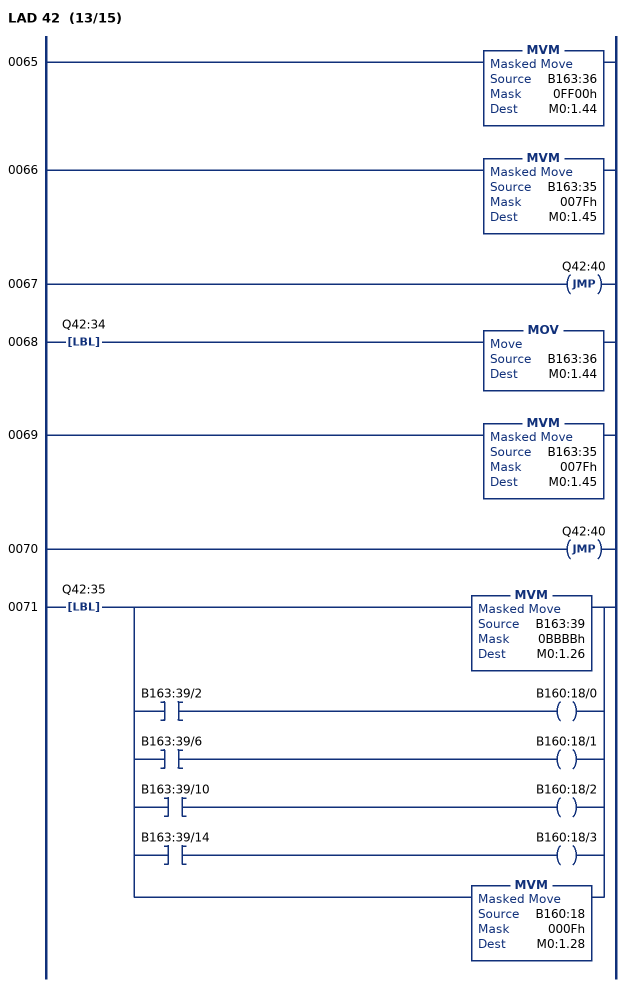
% Rung: 65 %
SOR MVM B163:36 0FF00h M0:1.44 EOR
% Rung: 66 %
SOR MVM B163:35 007Fh M0:1.45 EOR
% Rung: 67 %
SOR JMP Q42:40 EOR
% Rung: 68 %
SOR LBL Q42:34 MOV B163:36 M0:1.44 EOR
% Rung: 69 %
SOR MVM B163:35 007Fh M0:1.45 EOR
% Rung: 70 %
SOR JMP Q42:40 EOR
% Rung: 71 %
SOR LBL Q42:35 BST MVM B163:39 0BBBBh M0:1.26 NXB XIC B163:39/2 OTE B160:18/0 NXB XIC B163:39/6 OTE B160:18/1 NXB XIC B163:39/10 OTE B160:18/2 NXB XIC B163:39/14 OTE B160:18/3 NXB MVM B160:18 000Fh M0:1.28 BND EOR

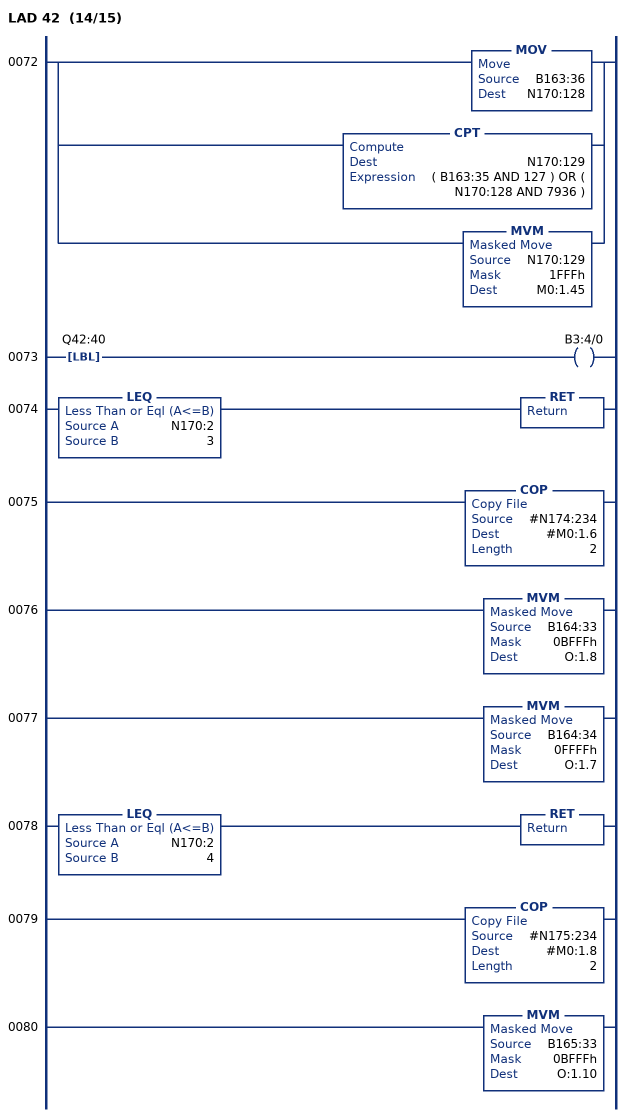
% Rung: 72 %
SOR BST MOV B163:36 N170:128 NXB CPT N170:129 " ( B163:35 AND 127 ) OR ( N170:128 AND 7936 ) " NXB MVM N170:129 1FFFh M0:1.45 BND EOR
% Rung: 73 %
SOR LBL Q42:40 OTE B3:4/0 EOR
% Rung: 74 %
SOR LEQ N170:2 3 RET EOR
% Rung: 75 %
SOR COP #N174:234 #M0:1.6 2 EOR
% Rung: 76 %
SOR MVM B164:33 0BFFFh O:1.8 EOR
% Rung: 77 %
SOR MVM B164:34 0FFFFh O:1.7 EOR
% Rung: 78 %
SOR LEQ N170:2 4 RET EOR
% Rung: 79 %
SOR COP #N175:234 #M0:1.8 2 EOR
% Rung: 80 %
SOR MVM B165:33 0BFFFh O:1.10 EOR

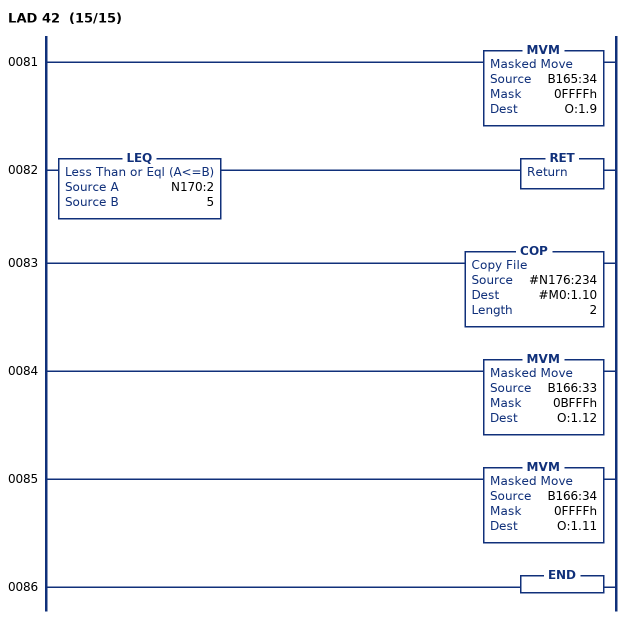
% Rung: 81 %
SOR MVM B165:34 0FFFFh O:1.9 EOR
% Rung: 82 %
SOR LEQ N170:2 5 RET EOR
% Rung: 83 %
SOR COP #N176:234 #M0:1.10 2 EOR
% Rung: 84 %
SOR MVM B166:33 0BFFFh O:1.12 EOR
% Rung: 85 %
SOR MVM B166:34 0FFFFh O:1.11 EOR
% Rung: 86 %
SOR END EOR

LADDER 43
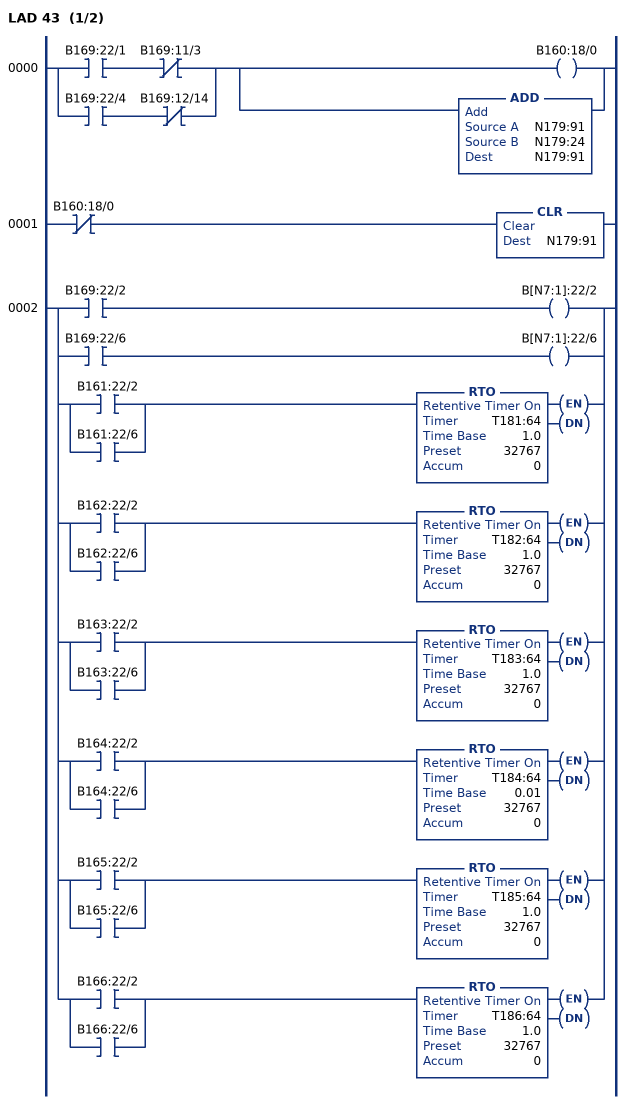
% Rung: 0 %
SOR BST XIC B169:22/1 XIO B169:11/3 NXB XIC B169:22/4 XIO B169:12/14 BND BST OTE B160:18/0 NXB ADD N179:91 N179:24 N179:91 BND EOR
% Rung: 1 %
SOR XIO B160:18/0 CLR N179:91 EOR
% Rung: 2 %
SOR BST BST XIC B169:22/2 OTE B[N7:1]:22/2 NXB XIC B169:22/6 OTE B[N7:1]:22/6 BND NXB BST XIC B161:22/2 NXB XIC B161:22/6 BND RTO T181:64 1.0 32767 0 NXB BST XIC B162:22/2 NXB XIC B162:22/6 BND RTO T182:64 1.0 32767 0 NXB BST XIC B163:22/2 NXB XIC B163:22/6 BND RTO T183:64 1.0 32767 0 NXB BST XIC B164:22/2 NXB XIC B164:22/6 BND RTO T184:64 0.01 32767 0 NXB BST XIC B165:22/2 NXB XIC B165:22/6 BND RTO T185:64 1.0 32767 0 NXB BST XIC B166:22/2 NXB XIC B166:22/6 BND RTO T186:64 1.0 32767 0 BND EOR

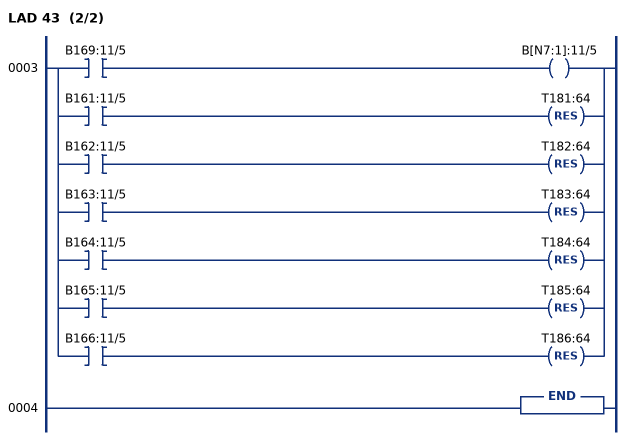
% Rung: 3 %
SOR BST XIC B169:11/5 OTE B[N7:1]:11/5 NXB XIC B161:11/5 RES T181:64 NXB XIC B162:11/5 RES T182:64 NXB XIC B163:11/5 RES T183:64 NXB XIC B164:11/5 RES T184:64 NXB XIC B165:11/5 RES T185:64 NXB XIC B166:11/5 RES T186:64 BND EOR
% Rung: 4 %
SOR END EOR

LADDER 44
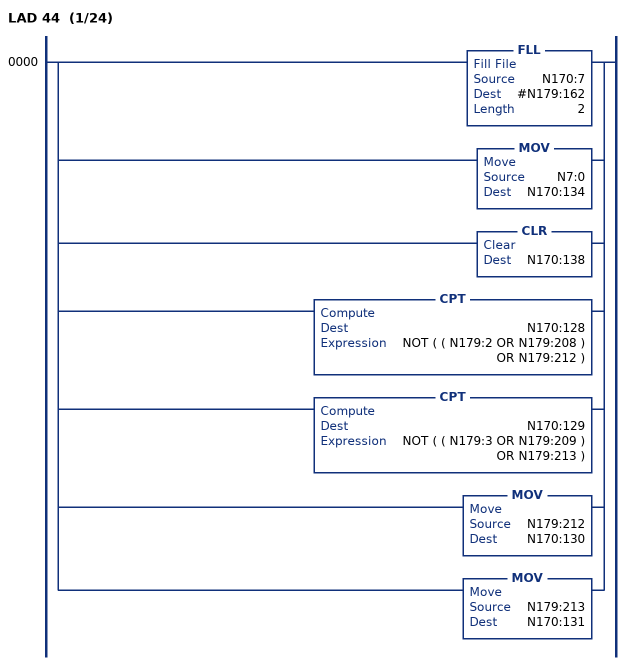
% Rung: 0 %
SOR BST FLL N170:7 #N179:162 2 NXB MOV N7:0 N170:134 NXB CLR N170:138 NXB CPT N170:128 " NOT ( ( N179:2 OR N179:208 ) OR N179:212 ) " NXB CPT N170:129 " NOT ( ( N179:3 OR N179:209 ) OR N179:213 ) " NXB MOV N179:212 N170:130 NXB MOV N179:213 N170:131 BND EOR

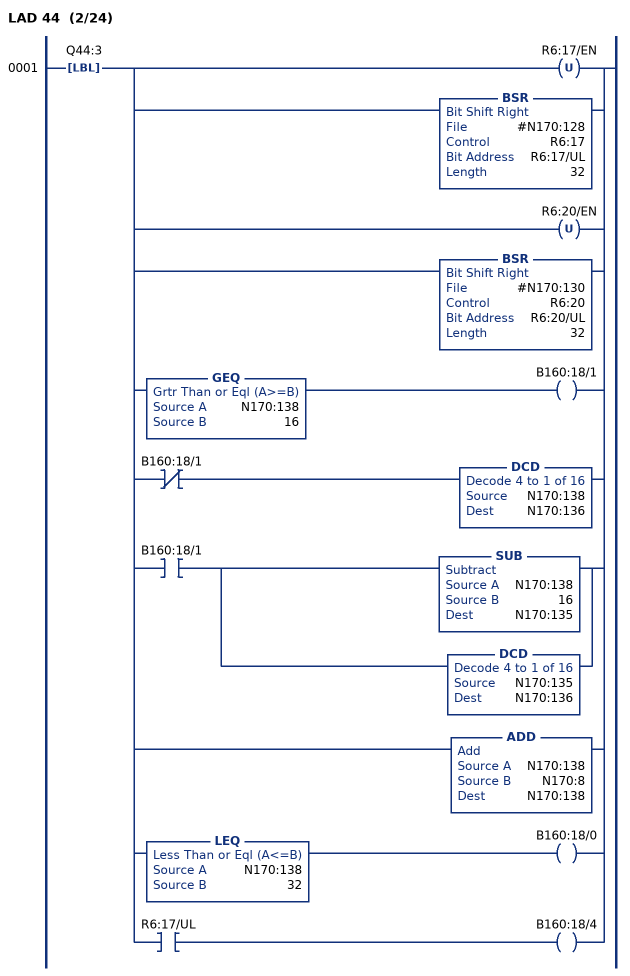
% Rung: 1 %
SOR LBL Q44:3 BST BST OTU R6:17/EN NXB BSR #N170:128 R6:17 R6:17/UL 32 BND NXB BST OTU R6:20/EN NXB BSR #N170:130 R6:20 R6:20/UL 32 BND NXB GEQ N170:138 16 OTE B160:18/1 NXB XIO B160:18/1 DCD N170:138 N170:136 NXB XIC B160:18/1 BST SUB N170:138 16 N170:135 NXB DCD N170:135 N170:136 BND NXB ADD N170:138 N170:8 N170:138 NXB LEQ N170:138 32 OTE B160:18/0 NXB XIC R6:17/UL OTE B160:18/4 BND EOR

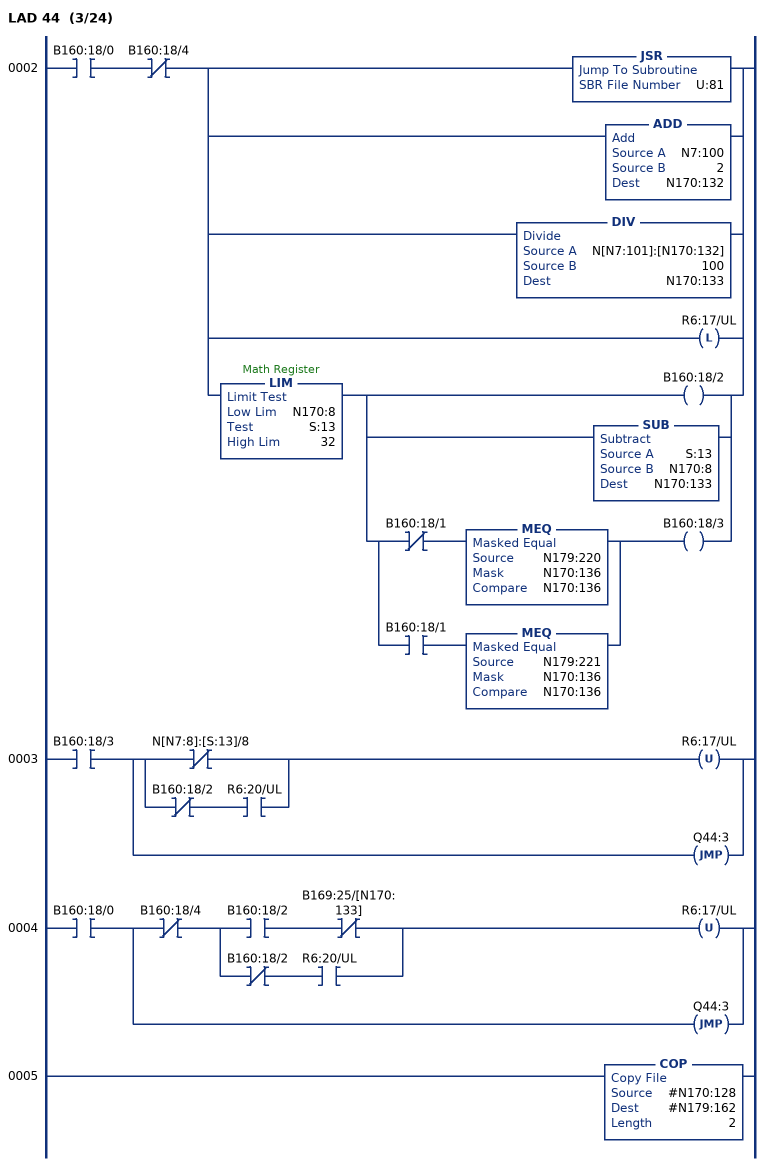
% Rung: 2 %
SOR XIC B160:18/0 XIO B160:18/4 BST JSR U:81 NXB ADD N7:100 2 N170:132 NXB DIV N[N7:101]:[N170:132] 100 N170:133 NXB OTL R6:17/UL NXB LIM N170:8 S:13 32 BST OTE B160:18/2 NXB SUB S:13 N170:8 N170:133 NXB BST XIO B160:18/1 MEQ N179:220 N170:136 N170:136 NXB XIC B160:18/1 MEQ N179:221 N170:136 N170:136 BND OTE B160:18/3 BND BND EOR
%   S:13  "Math Register" %
% Rung: 3 %
SOR XIC B160:18/3 BST BST XIO N[N7:8]:[S:13]/8 NXB XIO B160:18/2 XIC R6:20/UL BND OTU R6:17/UL NXB JMP Q44:3 BND EOR
%   S:13  "Math Register" %
% Rung: 4 %
SOR XIC B160:18/0 BST XIO B160:18/4 BST XIC B160:18/2 XIO B169:25/[N170:133] NXB XIO B160:18/2 XIC R6:20/UL BND OTU R6:17/UL NXB JMP Q44:3 BND EOR
% Rung: 5 %
SOR COP #N170:128 #N179:162 2 EOR

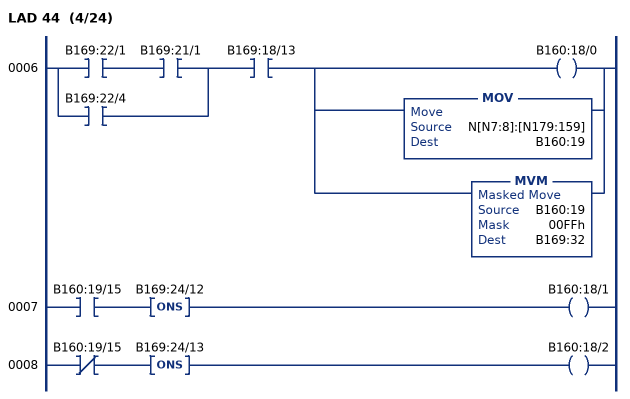
% Rung: 6 %
SOR BST XIC B169:22/1 XIC B169:21/1 NXB XIC B169:22/4 BND XIC B169:18/13 BST OTE B160:18/0 NXB MOV N[N7:8]:[N179:159] B160:19 NXB MVM B160:19 00FFh B169:32 BND EOR
% Rung: 7 %
SOR XIC B160:19/15 OSR B169:24/12 OTE B160:18/1 EOR
% Rung: 8 %
SOR XIO B160:19/15 OSR B169:24/13 OTE B160:18/2 EOR

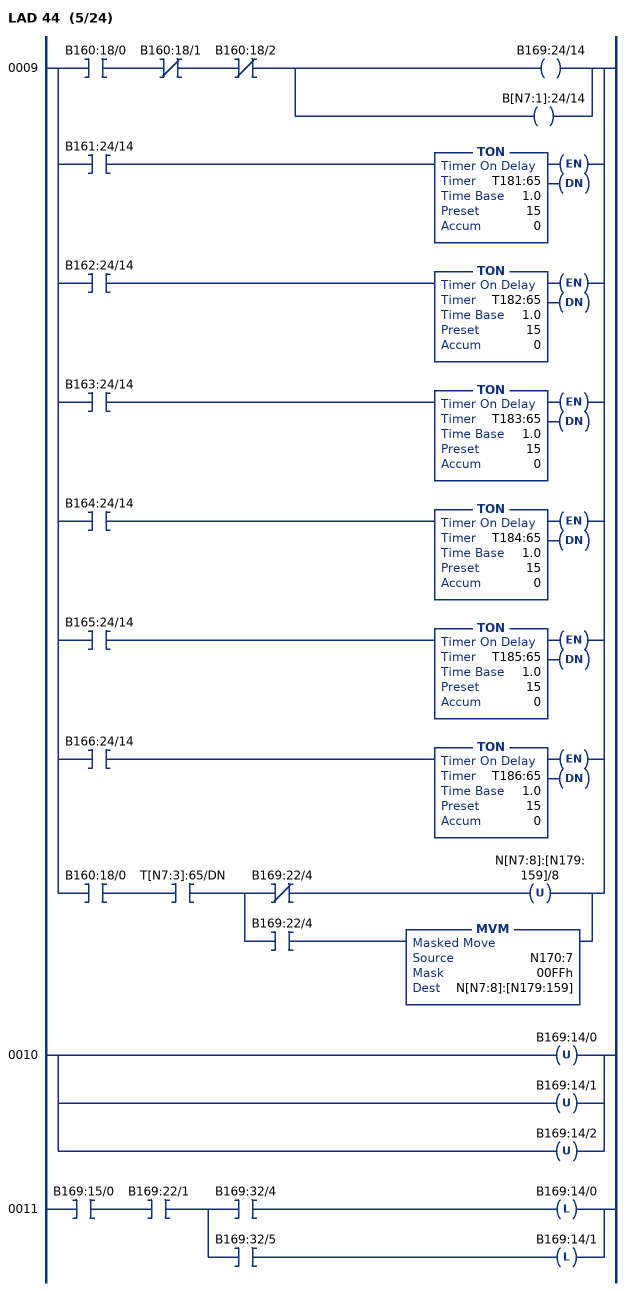
% Rung: 9 %
SOR BST BST XIC B160:18/0 XIO B160:18/1 XIO B160:18/2 BST OTE B169:24/14 NXB OTE B[N7:1]:24/14 BND NXB XIC B161:24/14 TON T181:65 1.0 15 0 NXB XIC B162:24/14 TON T182:65 1.0 15 0 NXB XIC B163:24/14 TON T183:65 1.0 15 0 NXB XIC B164:24/14 TON T184:65 1.0 15 0 NXB XIC B165:24/14 TON T185:65 1.0 15 0 NXB XIC B166:24/14 TON T186:65 1.0 15 0 BND NXB XIC B160:18/0 XIC T[N7:3]:65/DN BST XIO B169:22/4 OTU N[N7:8]:[N179:159]/8 NXB XIC B169:22/4 MVM N170:7 00FFh N[N7:8]:[N179:159] BND BND EOR
% Rung: 10 %
SOR BST OTU B169:14/0 NXB OTU B169:14/1 NXB OTU B169:14/2 BND EOR
% Rung: 11 %
SOR XIC B169:15/0 XIC B169:22/1 BST XIC B169:32/4 OTL B169:14/0 NXB XIC B169:32/5 OTL B169:14/1 BND EOR

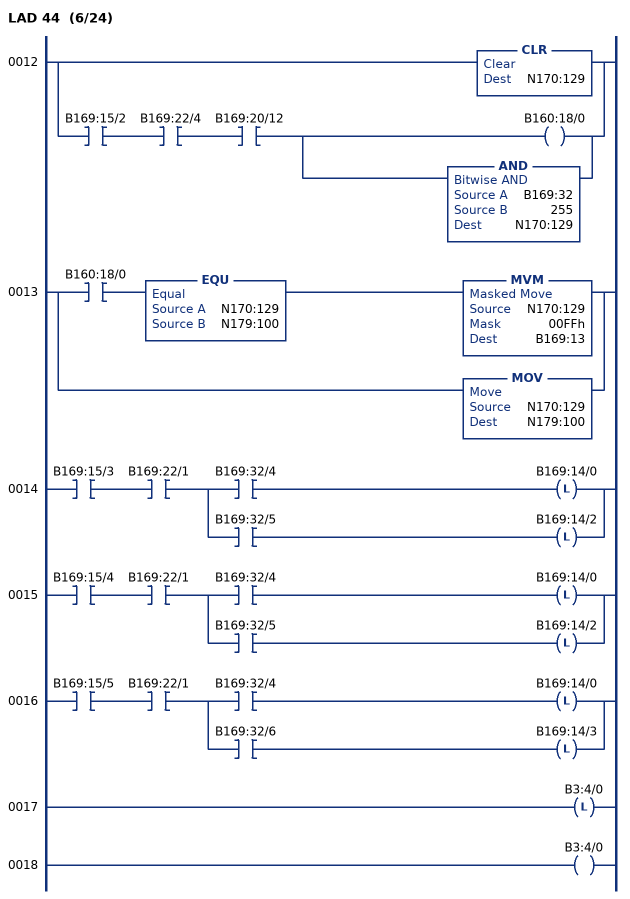
% Rung: 12 %
SOR BST CLR N170:129 NXB XIC B169:15/2 XIC B169:22/4 XIC B169:20/12 BST OTE B160:18/0 NXB AND B169:32 255 N170:129 BND BND EOR
% Rung: 13 %
SOR BST XIC B160:18/0 EQU N170:129 N179:100 MVM N170:129 00FFh B169:13 NXB MOV N170:129 N179:100 BND EOR
% Rung: 14 %
SOR XIC B169:15/3 XIC B169:22/1 BST XIC B169:32/4 OTL B169:14/0 NXB XIC B169:32/5 OTL B169:14/2 BND EOR
% Rung: 15 %
SOR XIC B169:15/4 XIC B169:22/1 BST XIC B169:32/4 OTL B169:14/0 NXB XIC B169:32/5 OTL B169:14/2 BND EOR
% Rung: 16 %
SOR XIC B169:15/5 XIC B169:22/1 BST XIC B169:32/4 OTL B169:14/0 NXB XIC B169:32/6 OTL B169:14/3 BND EOR
% Rung: 17 %
SOR OTL B3:4/0 EOR
% Rung: 18 %
SOR OTE B3:4/0 EOR

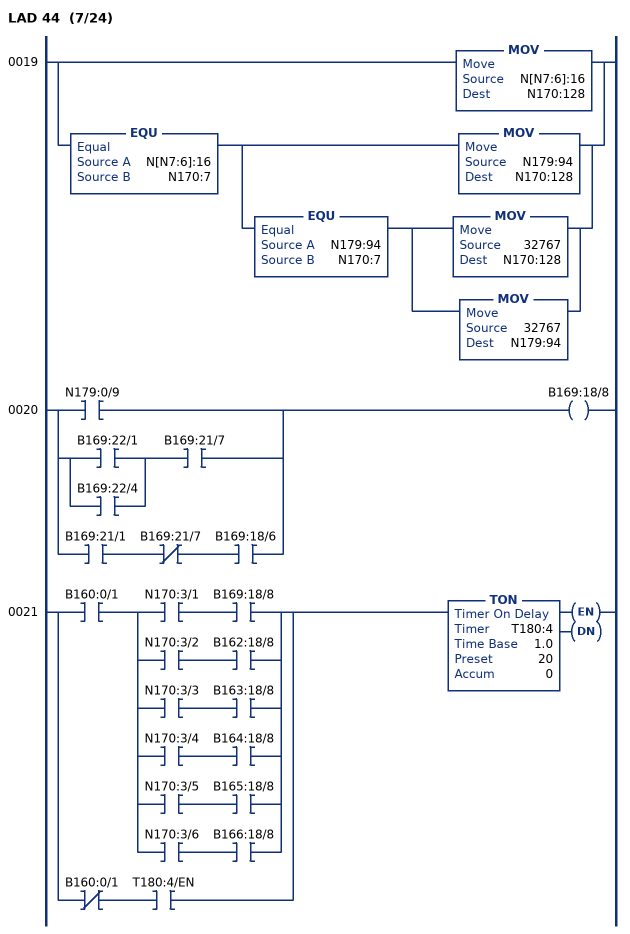
% Rung: 19 %
SOR BST MOV N[N7:6]:16 N170:128 NXB EQU N[N7:6]:16 N170:7 BST MOV N179:94 N170:128 NXB EQU N179:94 N170:7 BST MOV 32767 N170:128 NXB MOV 32767 N179:94 BND BND BND EOR
% Rung: 20 %
SOR BST XIC N179:0/9 NXB BST XIC B169:22/1 NXB XIC B169:22/4 BND XIC B169:21/7 NXB XIC B169:21/1 XIO B169:21/7 XIC B169:18/6 BND OTE B169:18/8 EOR
% Rung: 21 %
SOR BST XIC B160:0/1 BST XIC N170:3/1 XIC B169:18/8 NXB XIC N170:3/2 XIC B162:18/8 NXB XIC N170:3/3 XIC B163:18/8 NXB XIC N170:3/4 XIC B164:18/8 NXB XIC N170:3/5 XIC B165:18/8 NXB XIC N170:3/6 XIC B166:18/8 BND NXB XIO B160:0/1 XIC T180:4/EN BND TON T180:4 1.0 20 0 EOR

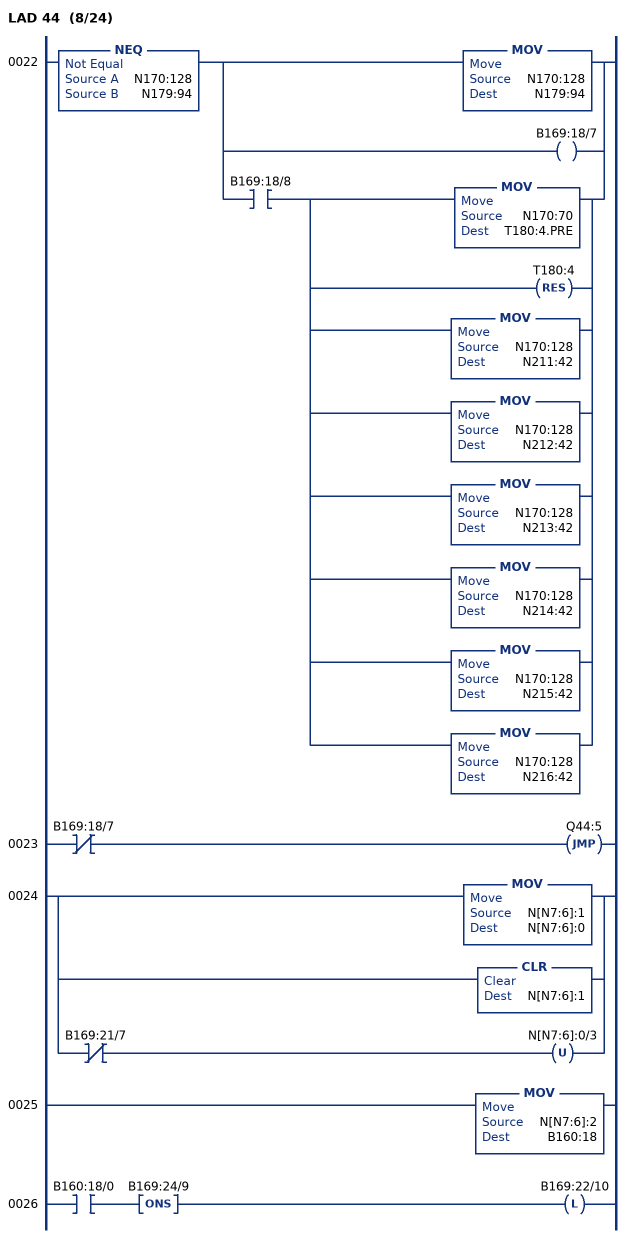
% Rung: 22 %
SOR NEQ N170:128 N179:94 BST MOV N170:128 N179:94 NXB OTE B169:18/7 NXB XIC B169:18/8 BST MOV N170:70 T180:4.PRE NXB RES T180:4 NXB MOV N170:128 N211:42 NXB MOV N170:128 N212:42 NXB MOV N170:128 N213:42 NXB MOV N170:128 N214:42 NXB MOV N170:128 N215:42 NXB MOV N170:128 N216:42 BND BND EOR
% Rung: 23 %
SOR XIO B169:18/7 JMP Q44:5 EOR
% Rung: 24 %
SOR BST MOV N[N7:6]:1 N[N7:6]:0 NXB CLR N[N7:6]:1 NXB XIO B169:21/7 OTU N[N7:6]:0/3 BND EOR
% Rung: 25 %
SOR MOV N[N7:6]:2 B160:18 EOR
% Rung: 26 %
SOR XIC B160:18/0 OSR B169:24/9 OTL B169:22/10 EOR

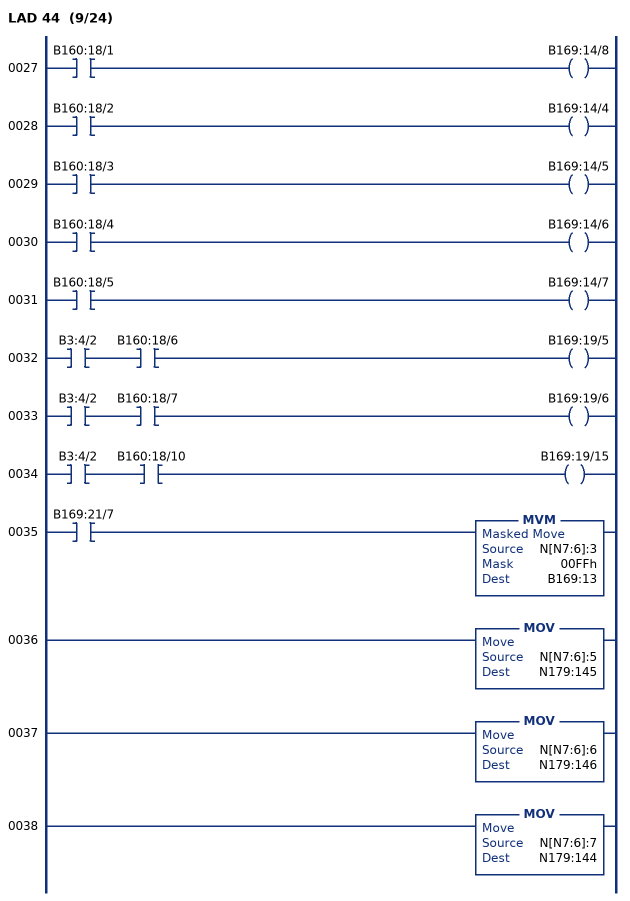
% Rung: 27 %
SOR XIC B160:18/1 OTE B169:14/8 EOR
% Rung: 28 %
SOR XIC B160:18/2 OTE B169:14/4 EOR
% Rung: 29 %
SOR XIC B160:18/3 OTE B169:14/5 EOR
% Rung: 30 %
SOR XIC B160:18/4 OTE B169:14/6 EOR
% Rung: 31 %
SOR XIC B160:18/5 OTE B169:14/7 EOR
% Rung: 32 %
SOR XIC B3:4/2 XIC B160:18/6 OTE B169:19/5 EOR
% Rung: 33 %
SOR XIC B3:4/2 XIC B160:18/7 OTE B169:19/6 EOR
% Rung: 34 %
SOR XIC B3:4/2 XIC B160:18/10 OTE B169:19/15 EOR
% Rung: 35 %
SOR XIC B169:21/7 MVM N[N7:6]:3 00FFh B169:13 EOR
% Rung: 36 %
SOR MOV N[N7:6]:5 N179:145 EOR
% Rung: 37 %
SOR MOV N[N7:6]:6 N179:146 EOR
% Rung: 38 %
SOR MOV N[N7:6]:7 N179:144 EOR

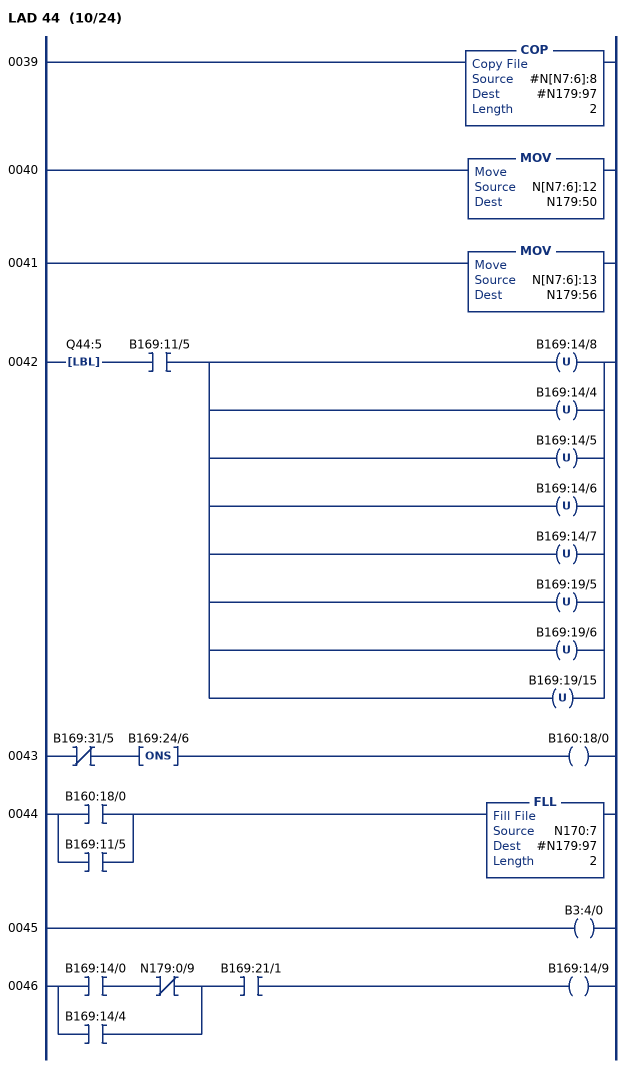
% Rung: 39 %
SOR COP #N[N7:6]:8 #N179:97 2 EOR
% Rung: 40 %
SOR MOV N[N7:6]:12 N179:50 EOR
% Rung: 41 %
SOR MOV N[N7:6]:13 N179:56 EOR
% Rung: 42 %
SOR LBL Q44:5 XIC B169:11/5 BST OTU B169:14/8 NXB OTU B169:14/4 NXB OTU B169:14/5 NXB OTU B169:14/6 NXB OTU B169:14/7 NXB OTU B169:19/5 NXB OTU B169:19/6 NXB OTU B169:19/15 BND EOR
% Rung: 43 %
SOR XIO B169:31/5 OSR B169:24/6 OTE B160:18/0 EOR
% Rung: 44 %
SOR BST XIC B160:18/0 NXB XIC B169:11/5 BND FLL N170:7 #N179:97 2 EOR
% Rung: 45 %
SOR OTE B3:4/0 EOR
% Rung: 46 %
SOR BST XIC B169:14/0 XIO N179:0/9 NXB XIC B169:14/4 BND XIC B169:21/1 OTE B169:14/9 EOR

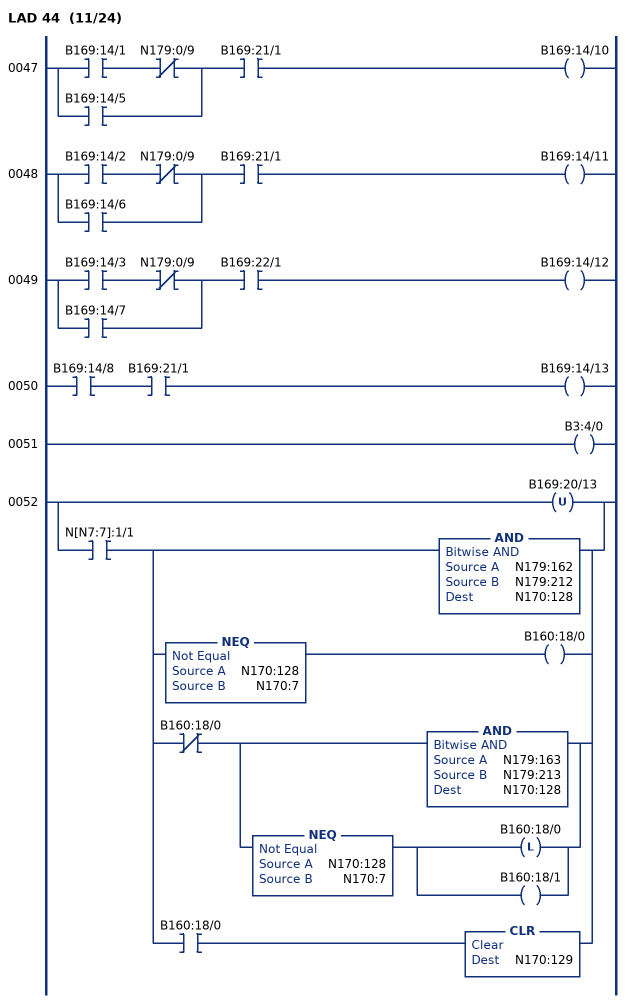
% Rung: 47 %
SOR BST XIC B169:14/1 XIO N179:0/9 NXB XIC B169:14/5 BND XIC B169:21/1 OTE B169:14/10 EOR
% Rung: 48 %
SOR BST XIC B169:14/2 XIO N179:0/9 NXB XIC B169:14/6 BND XIC B169:21/1 OTE B169:14/11 EOR
% Rung: 49 %
SOR BST XIC B169:14/3 XIO N179:0/9 NXB XIC B169:14/7 BND XIC B169:22/1 OTE B169:14/12 EOR
% Rung: 50 %
SOR XIC B169:14/8 XIC B169:21/1 OTE B169:14/13 EOR
% Rung: 51 %
SOR OTE B3:4/0 EOR
% Rung: 52 %
SOR BST OTU B169:20/13 NXB XIC N[N7:7]:1/1 BST AND N179:162 N179:212 N170:128 NXB NEQ N170:128 N170:7 OTE B160:18/0 NXB XIO B160:18/0 BST AND N179:163 N179:213 N170:128 NXB NEQ N170:128 N170:7 BST OTL B160:18/0 NXB OTE B160:18/1 BND BND NXB XIC B160:18/0 CLR N170:129 BND BND EOR

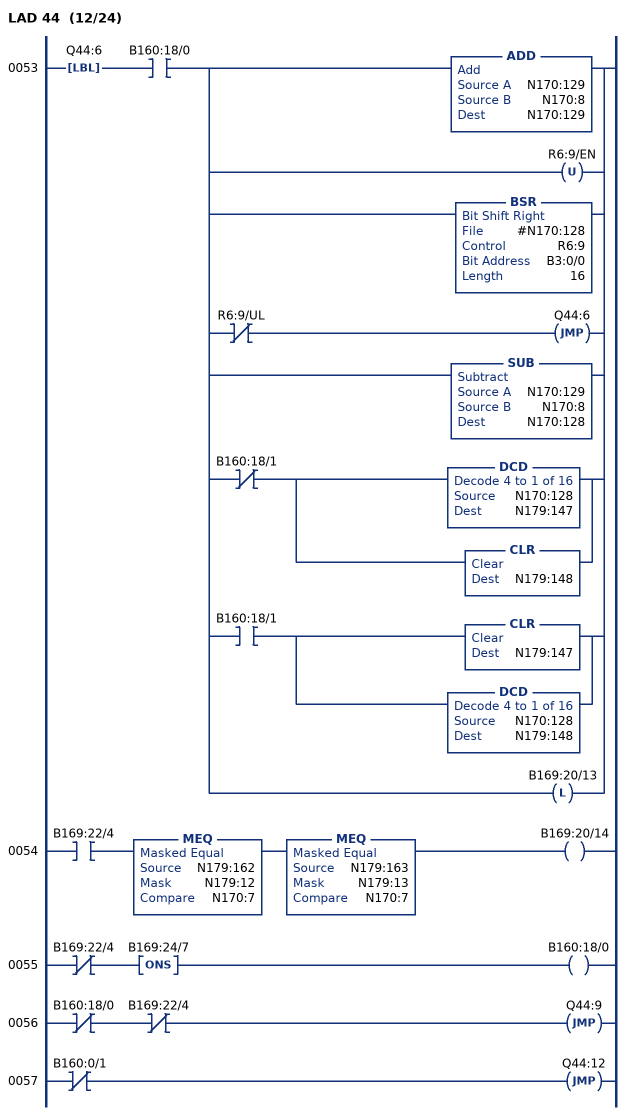
% Rung: 53 %
SOR LBL Q44:6 XIC B160:18/0 BST ADD N170:129 N170:8 N170:129 NXB OTU R6:9/EN NXB BSR #N170:128 R6:9 B3:0/0 16 NXB XIO R6:9/UL JMP Q44:6 NXB SUB N170:129 N170:8 N170:128 NXB XIO B160:18/1 BST DCD N170:128 N179:147 NXB CLR N179:148 BND NXB XIC B160:18/1 BST CLR N179:147 NXB DCD N170:128 N179:148 BND NXB OTL B169:20/13 BND EOR
% Rung: 54 %
SOR XIC B169:22/4 MEQ N179:162 N179:12 N170:7 MEQ N179:163 N179:13 N170:7 OTE B169:20/14 EOR
% Rung: 55 %
SOR XIO B169:22/4 OSR B169:24/7 OTE B160:18/0 EOR
% Rung: 56 %
SOR XIO B160:18/0 XIO B169:22/4 JMP Q44:9 EOR
% Rung: 57 %
SOR XIO B160:0/1 JMP Q44:12 EOR

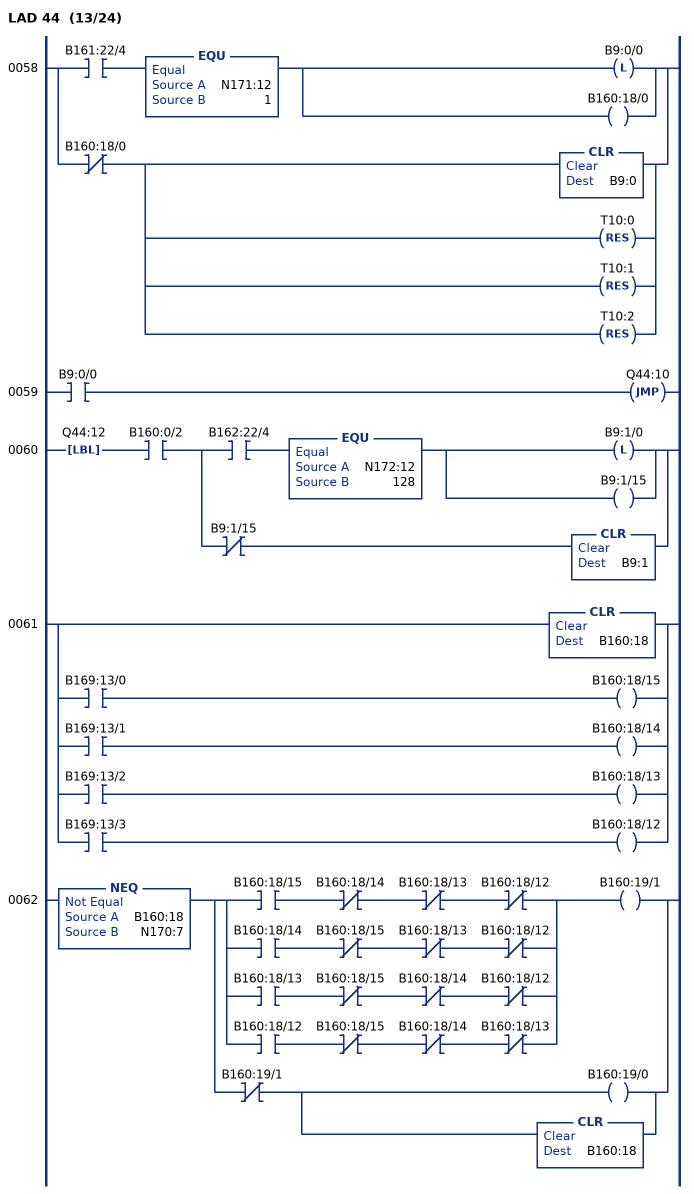
% Rung: 58 %
SOR BST XIC B161:22/4 EQU N171:12 1 BST OTL B9:0/0 NXB OTE B160:18/0 BND NXB XIO B160:18/0 BST CLR B9:0 NXB BST RES T10:0 NXB RES T10:1 NXB RES T10:2 BND BND BND EOR
% Rung: 59 %
SOR XIC B9:0/0 JMP Q44:10 EOR
% Rung: 60 %
SOR LBL Q44:12 XIC B160:0/2 BST XIC B162:22/4 EQU N172:12 128 BST OTL B9:1/0 NXB OTE B9:1/15 BND NXB XIO B9:1/15 CLR B9:1 BND EOR
% Rung: 61 %
SOR BST CLR B160:18 NXB XIC B169:13/0 OTE B160:18/15 NXB XIC B169:13/1 OTE B160:18/14 NXB XIC B169:13/2 OTE B160:18/13 NXB XIC B169:13/3 OTE B160:18/12 BND EOR
% Rung: 62 %
SOR NEQ B160:18 N170:7 BST BST XIC B160:18/15 XIO B160:18/14 XIO B160:18/13 XIO B160:18/12 NXB XIC B160:18/14 XIO B160:18/15 XIO B160:18/13 XIO B160:18/12 NXB XIC B160:18/13 XIO B160:18/15 XIO B160:18/14 XIO B160:18/12 NXB XIC B160:18/12 XIO B160:18/15 XIO B160:18/14 XIO B160:18/13 BND OTE B160:19/1 NXB XIO B160:19/1 BST OTE B160:19/0 NXB CLR B160:18 BND BND EOR

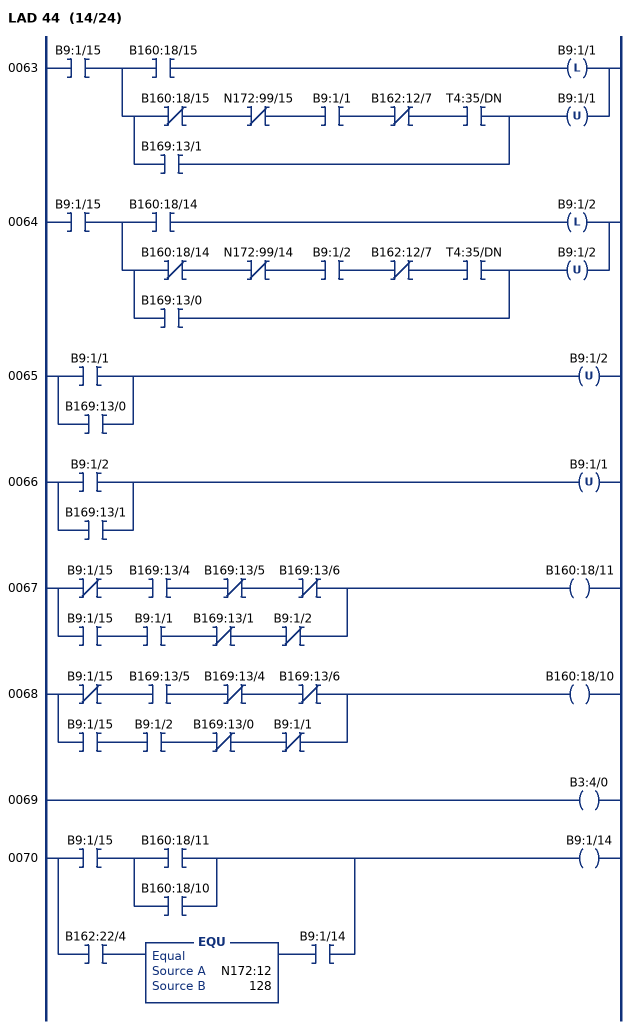
% Rung: 63 %
SOR XIC B9:1/15 BST XIC B160:18/15 OTL B9:1/1 NXB BST XIO B160:18/15 XIO N172:99/15 XIC B9:1/1 XIO B162:12/7 XIC T4:35/DN NXB XIC B169:13/1 BND OTU B9:1/1 BND EOR
% Rung: 64 %
SOR XIC B9:1/15 BST XIC B160:18/14 OTL B9:1/2 NXB BST XIO B160:18/14 XIO N172:99/14 XIC B9:1/2 XIO B162:12/7 XIC T4:35/DN NXB XIC B169:13/0 BND OTU B9:1/2 BND EOR
% Rung: 65 %
SOR BST XIC B9:1/1 NXB XIC B169:13/0 BND OTU B9:1/2 EOR
% Rung: 66 %
SOR BST XIC B9:1/2 NXB XIC B169:13/1 BND OTU B9:1/1 EOR
% Rung: 67 %
SOR BST XIO B9:1/15 XIC B169:13/4 XIO B169:13/5 XIO B169:13/6 NXB XIC B9:1/15 XIC B9:1/1 XIO B169:13/1 XIO B9:1/2 BND OTE B160:18/11 EOR
% Rung: 68 %
SOR BST XIO B9:1/15 XIC B169:13/5 XIO B169:13/4 XIO B169:13/6 NXB XIC B9:1/15 XIC B9:1/2 XIO B169:13/0 XIO B9:1/1 BND OTE B160:18/10 EOR
% Rung: 69 %
SOR OTE B3:4/0 EOR
% Rung: 70 %
SOR BST XIC B9:1/15 BST XIC B160:18/11 NXB XIC B160:18/10 BND NXB XIC B162:22/4 EQU N172:12 128 XIC B9:1/14 BND OTE B9:1/14 EOR

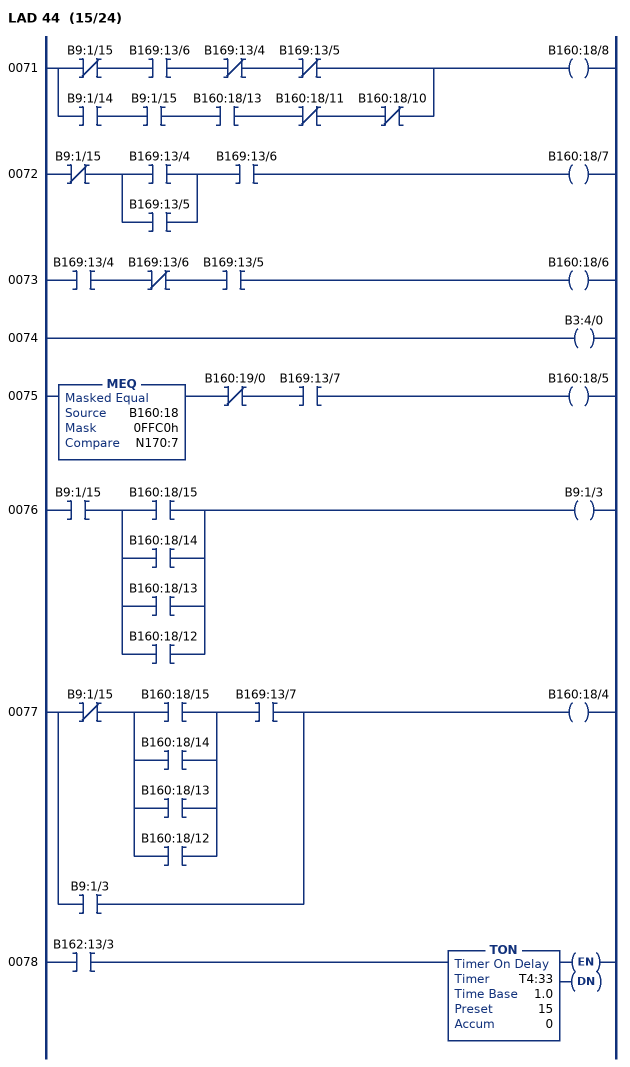
% Rung: 71 %
SOR BST XIO B9:1/15 XIC B169:13/6 XIO B169:13/4 XIO B169:13/5 NXB XIC B9:1/14 XIC B9:1/15 XIC B160:18/13 XIO B160:18/11 XIO B160:18/10 BND OTE B160:18/8 EOR
% Rung: 72 %
SOR XIO B9:1/15 BST XIC B169:13/4 NXB XIC B169:13/5 BND XIC B169:13/6 OTE B160:18/7 EOR
% Rung: 73 %
SOR XIC B169:13/4 XIO B169:13/6 XIC B169:13/5 OTE B160:18/6 EOR
% Rung: 74 %
SOR OTE B3:4/0 EOR
% Rung: 75 %
SOR MEQ B160:18 0FFC0h N170:7 XIO B160:19/0 XIC B169:13/7 OTE B160:18/5 EOR
% Rung: 76 %
SOR XIC B9:1/15 BST XIC B160:18/15 NXB XIC B160:18/14 NXB XIC B160:18/13 NXB XIC B160:18/12 BND OTE B9:1/3 EOR
% Rung: 77 %
SOR BST XIO B9:1/15 BST XIC B160:18/15 NXB XIC B160:18/14 NXB XIC B160:18/13 NXB XIC B160:18/12 BND XIC B169:13/7 NXB XIC B9:1/3 BND OTE B160:18/4 EOR
% Rung: 78 %
SOR XIC B162:13/3 TON T4:33 1.0 15 0 EOR

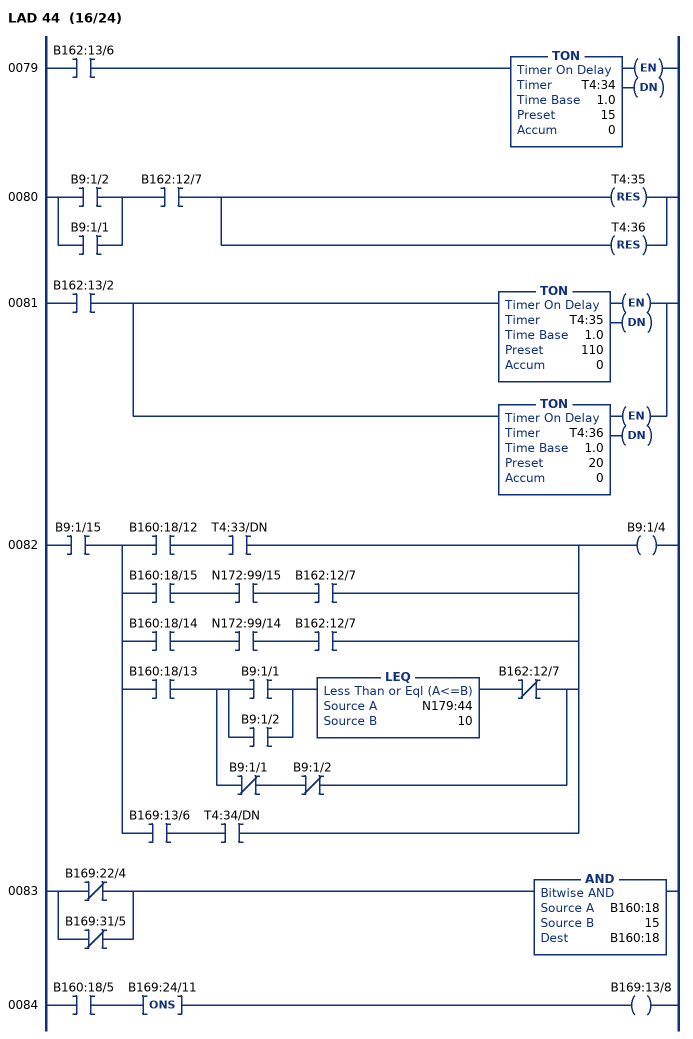
% Rung: 79 %
SOR XIC B162:13/6 TON T4:34 1.0 15 0 EOR
% Rung: 80 %
SOR BST XIC B9:1/2 NXB XIC B9:1/1 BND XIC B162:12/7 BST RES T4:35 NXB RES T4:36 BND EOR
% Rung: 81 %
SOR XIC B162:13/2 BST TON T4:35 1.0 110 0 NXB TON T4:36 1.0 20 0 BND EOR
% Rung: 82 %
SOR XIC B9:1/15 BST XIC B160:18/12 XIC T4:33/DN NXB XIC B160:18/15 XIC N172:99/15 XIC B162:12/7 NXB XIC B160:18/14 XIC N172:99/14 XIC B162:12/7 NXB XIC B160:18/13 BST BST XIC B9:1/1 NXB XIC B9:1/2 BND LEQ N179:44 10 XIO B162:12/7 NXB XIO B9:1/1 XIO B9:1/2 BND NXB XIC B169:13/6 XIC T4:34/DN BND OTE B9:1/4 EOR
% Rung: 83 %
SOR BST XIO B169:22/4 NXB XIO B169:31/5 BND AND B160:18 15 B160:18 EOR
% Rung: 84 %
SOR XIC B160:18/5 OSR B169:24/11 OTE B169:13/8 EOR

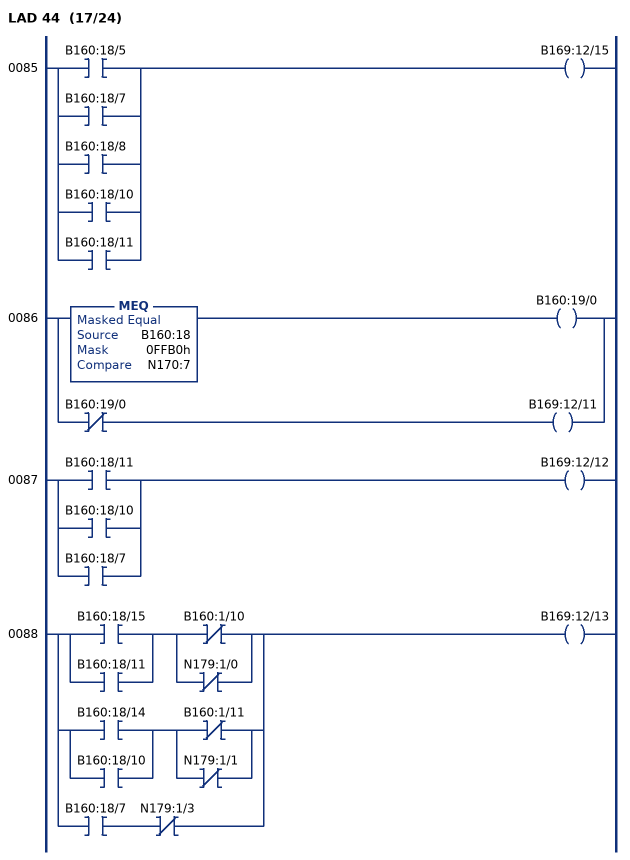
% Rung: 85 %
SOR BST XIC B160:18/5 NXB XIC B160:18/7 NXB XIC B160:18/8 NXB XIC B160:18/10 NXB XIC B160:18/11 BND OTE B169:12/15 EOR
% Rung: 86 %
SOR BST MEQ B160:18 0FFB0h N170:7 OTE B160:19/0 NXB XIO B160:19/0 OTE B169:12/11 BND EOR
% Rung: 87 %
SOR BST XIC B160:18/11 NXB XIC B160:18/10 NXB XIC B160:18/7 BND OTE B169:12/12 EOR
% Rung: 88 %
SOR BST BST XIC B160:18/15 NXB XIC B160:18/11 BND BST XIO B160:1/10 NXB XIO N179:1/0 BND NXB BST XIC B160:18/14 NXB XIC B160:18/10 BND BST XIO B160:1/11 NXB XIO N179:1/1 BND NXB XIC B160:18/7 XIO N179:1/3 BND OTE B169:12/13 EOR

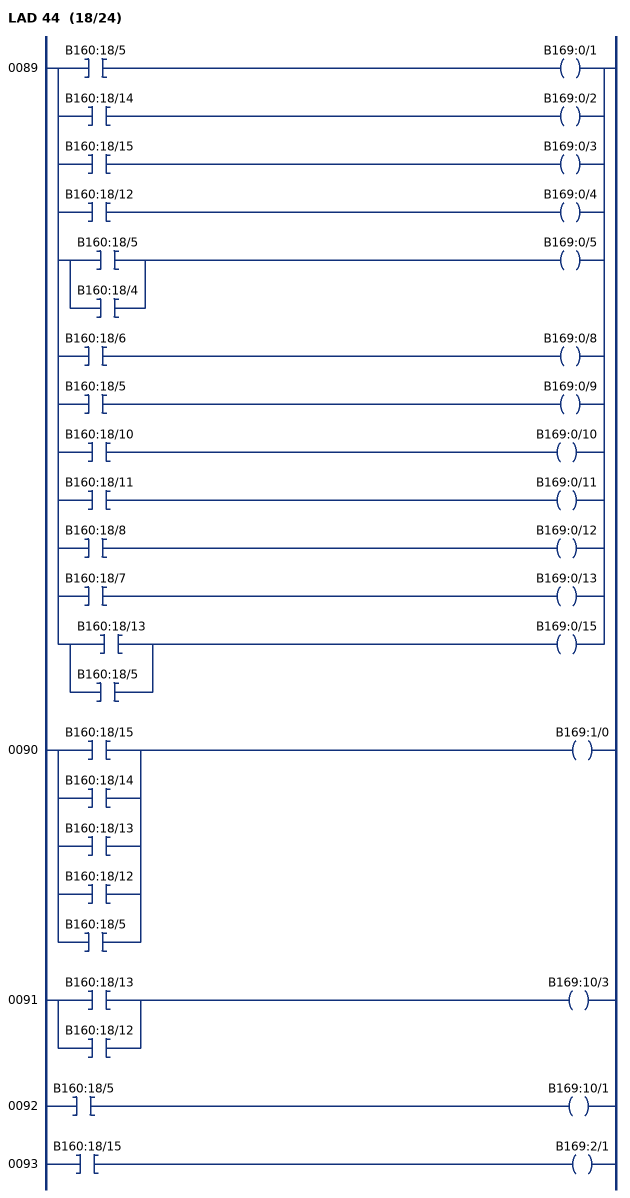
% Rung: 89 %
SOR BST XIC B160:18/5 OTE B169:0/1 NXB XIC B160:18/14 OTE B169:0/2 NXB XIC B160:18/15 OTE B169:0/3 NXB XIC B160:18/12 OTE B169:0/4 NXB BST XIC B160:18/5 NXB XIC B160:18/4 BND OTE B169:0/5 NXB XIC B160:18/6 OTE B169:0/8 NXB XIC B160:18/5 OTE B169:0/9 NXB XIC B160:18/10 OTE B169:0/10 NXB XIC B160:18/11 OTE B169:0/11 NXB XIC B160:18/8 OTE B169:0/12 NXB XIC B160:18/7 OTE B169:0/13 NXB BST XIC B160:18/13 NXB XIC B160:18/5 BND OTE B169:0/15 BND EOR
% Rung: 90 %
SOR BST XIC B160:18/15 NXB XIC B160:18/14 NXB XIC B160:18/13 NXB XIC B160:18/12 NXB XIC B160:18/5 BND OTE B169:1/0 EOR
% Rung: 91 %
SOR BST XIC B160:18/13 NXB XIC B160:18/12 BND OTE B169:10/3 EOR
% Rung: 92 %
SOR XIC B160:18/5 OTE B169:10/1 EOR
% Rung: 93 %
SOR XIC B160:18/15 OTE B169:2/1 EOR

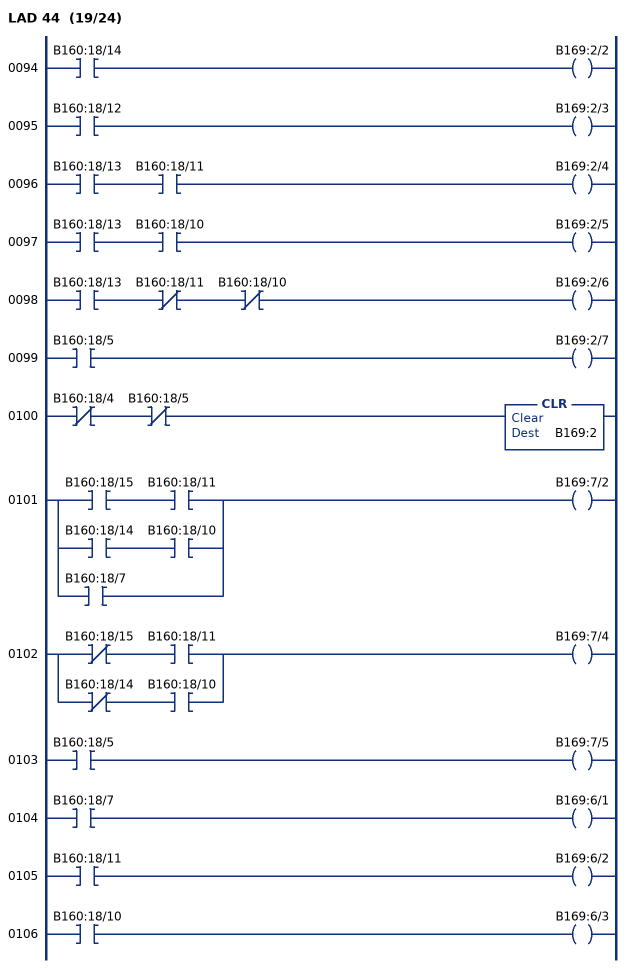
% Rung: 94 %
SOR XIC B160:18/14 OTE B169:2/2 EOR
% Rung: 95 %
SOR XIC B160:18/12 OTE B169:2/3 EOR
% Rung: 96 %
SOR XIC B160:18/13 XIC B160:18/11 OTE B169:2/4 EOR
% Rung: 97 %
SOR XIC B160:18/13 XIC B160:18/10 OTE B169:2/5 EOR
% Rung: 98 %
SOR XIC B160:18/13 XIO B160:18/11 XIO B160:18/10 OTE B169:2/6 EOR
% Rung: 99 %
SOR XIC B160:18/5 OTE B169:2/7 EOR
% Rung: 100 %
SOR XIO B160:18/4 XIO B160:18/5 CLR B169:2 EOR
% Rung: 101 %
SOR BST XIC B160:18/15 XIC B160:18/11 NXB XIC B160:18/14 XIC B160:18/10 NXB XIC B160:18/7 BND OTE B169:7/2 EOR
% Rung: 102 %
SOR BST XIO B160:18/15 XIC B160:18/11 NXB XIO B160:18/14 XIC B160:18/10 BND OTE B169:7/4 EOR
% Rung: 103 %
SOR XIC B160:18/5 OTE B169:7/5 EOR
% Rung: 104 %
SOR XIC B160:18/7 OTE B169:6/1 EOR
% Rung: 105 %
SOR XIC B160:18/11 OTE B169:6/2 EOR
% Rung: 106 %
SOR XIC B160:18/10 OTE B169:6/3 EOR

